(* CoDeSys 2.3.9.62 project: DrehtellerATN.pro *)
(* Libraries: Standard.lib, IecSfc.lib 2.6.14 10:37:46, SYSLIBCALLBACK.LIB *)

(* Global variable list: Global_Variables *)
VAR_GLOBAL
	Global_START: BOOL;
	K1: BOOL;
	K2: BOOL;
	Rechts: BOOL;
	Links: BOOL;
	Not_Aus: BOOL;
END_VAR

(* POU PLC_PRG, FBD *)
PROGRAM PLC_PRG
VAR
	Zweihand_Timer: TON;

END_VAR
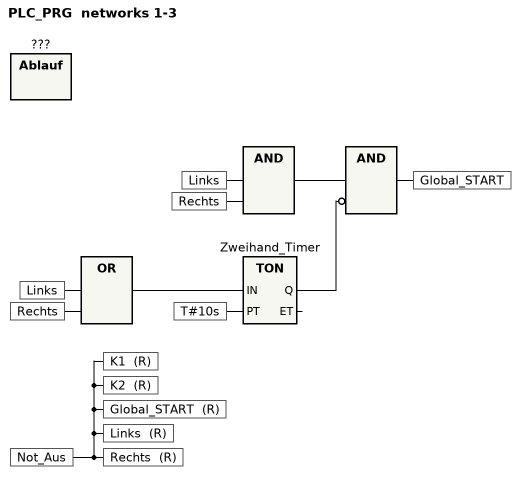
_FBD_ (* Function Block Diagram *)
NETWORK 1
	???:Ablauf()
NETWORK 2
	AND(AND(Links, Rechts), NOT Zweihand_Timer:TON(IN: OR(Links, Rechts), PT: T#10s)) => Global_START
NETWORK 3
	<<<<Not_Aus => R K1> => R K2> => R Global_START> => R Links> => R Rechts
_END_FBD_
(* the same logic as Structured Text *)
(* Network 1: see the listing above *)
(* Network 2 *)
Zweihand_Timer(IN := Links OR Rechts, PT := T#10s);
Global_START := (Links AND Rechts) AND NOT Zweihand_Timer.Q;
(* Network 3 *)
IF Not_Aus THEN K1 := FALSE; END_IF;
IF Not_Aus THEN K2 := FALSE; END_IF;
IF Not_Aus THEN Global_START := FALSE; END_IF;
IF Not_Aus THEN Links := FALSE; END_IF;
IF Not_Aus THEN Rechts := FALSE; END_IF;
END_PROGRAM

(* POU Ablauf, SFC *)
PROGRAM Ablauf
VAR
	angle:INT:=0;
	oben: BOOL:=TRUE;
	unten: BOOL;
	S1: BOOL:=TRUE;
	T1: BOOL;
	Timer1: TON;
	tor: INT;
	Rotate: BOOL:=FALSE;
END_VAR
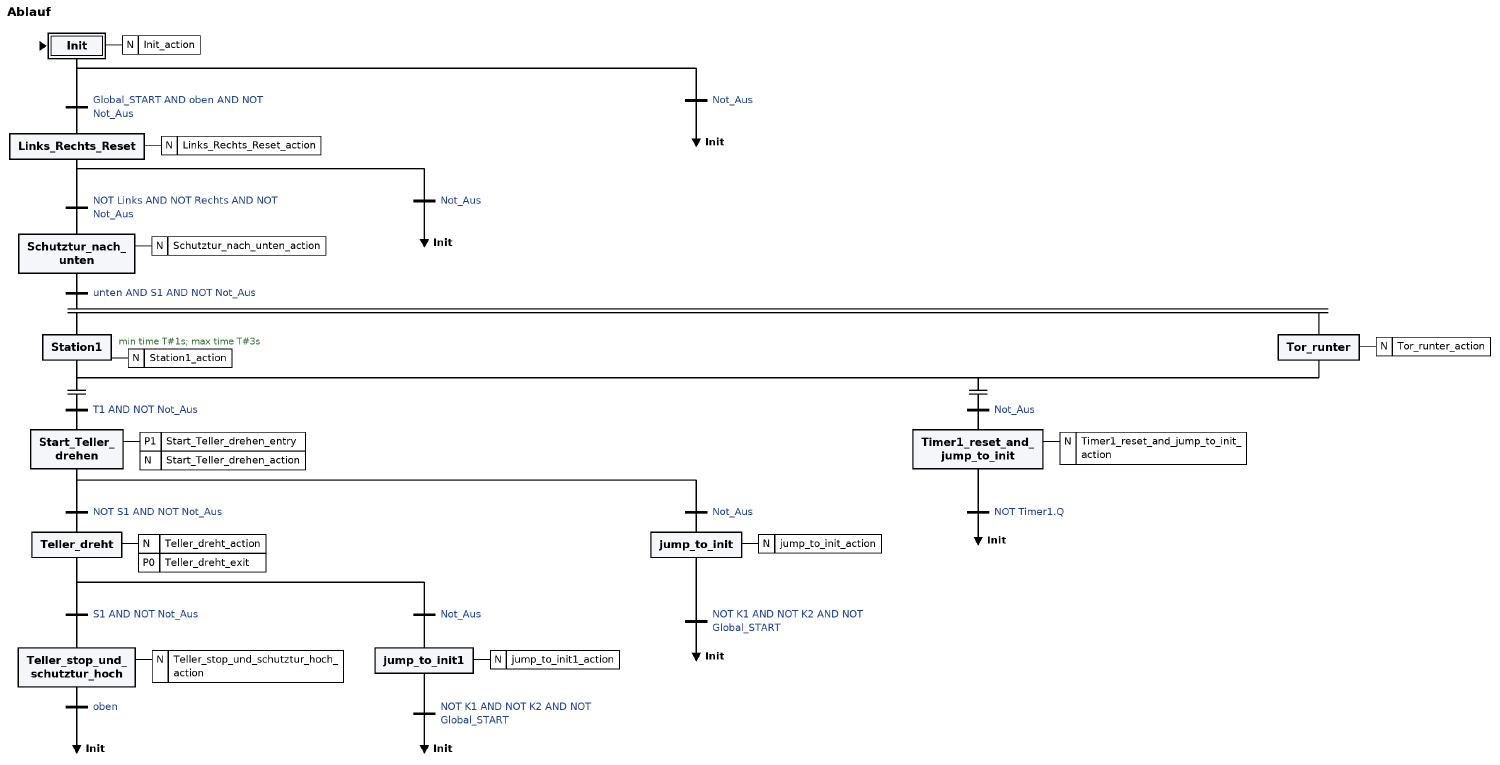
INITIAL_STEP Init:
	Init_action(N);
END_STEP
TRANSITION FROM Init TO Links_Rechts_Reset := Global_START AND oben AND NOT Not_Aus;
END_TRANSITION
TRANSITION FROM Init TO Init := Not_Aus;
END_TRANSITION
STEP Links_Rechts_Reset:
	Links_Rechts_Reset_action(N);
END_STEP
TRANSITION FROM Links_Rechts_Reset TO Schutztur_nach_unten := NOT Links AND NOT Rechts AND NOT Not_Aus;
END_TRANSITION
TRANSITION FROM Links_Rechts_Reset TO Init := Not_Aus;
END_TRANSITION
STEP Schutztur_nach_unten:
	Schutztur_nach_unten_action(N);
END_STEP
TRANSITION FROM Schutztur_nach_unten TO (Station1, Tor_runter) := unten AND S1 AND NOT Not_Aus;
END_TRANSITION
STEP Station1: (* min time T#1s; max time T#3s *)
	Station1_action(N);
END_STEP
STEP Tor_runter:
	Tor_runter_action(N);
END_STEP
TRANSITION FROM (Station1, Tor_runter) TO Start_Teller_drehen := T1 AND NOT Not_Aus;
END_TRANSITION
TRANSITION FROM (Station1, Tor_runter) TO Timer1_reset_and_jump_to_init := Not_Aus;
END_TRANSITION
STEP Timer1_reset_and_jump_to_init:
	Timer1_reset_and_jump_to_init_action(N);
END_STEP
TRANSITION FROM Timer1_reset_and_jump_to_init TO Init := NOT Timer1.Q;
END_TRANSITION
STEP Start_Teller_drehen:
	Start_Teller_drehen_entry(P1);
	Start_Teller_drehen_action(N);
END_STEP
TRANSITION FROM Start_Teller_drehen TO Teller_dreht := NOT S1 AND NOT Not_Aus;
END_TRANSITION
TRANSITION FROM Start_Teller_drehen TO jump_to_init := Not_Aus;
END_TRANSITION
STEP jump_to_init:
	jump_to_init_action(N);
END_STEP
TRANSITION FROM jump_to_init TO Init := NOT K1 AND NOT K2 AND NOT Global_START;
END_TRANSITION
STEP Teller_dreht:
	Teller_dreht_action(N);
	Teller_dreht_exit(P0);
END_STEP
TRANSITION FROM Teller_dreht TO Teller_stop_und_schutztur_hoch := S1 AND NOT Not_Aus;
END_TRANSITION
TRANSITION FROM Teller_dreht TO jump_to_init1 := Not_Aus;
END_TRANSITION
STEP jump_to_init1:
	jump_to_init1_action(N);
END_STEP
TRANSITION FROM jump_to_init1 TO Init := NOT K1 AND NOT K2 AND NOT Global_START;
END_TRANSITION
STEP Teller_stop_und_schutztur_hoch:
	Teller_stop_und_schutztur_hoch_action(N);
END_STEP
TRANSITION FROM Teller_stop_und_schutztur_hoch TO Init := oben;
END_TRANSITION

ACTION Init_action:
IF tor>0 THEN
tor:=tor-60;
S1:=TRUE;
END_IF
END_ACTION

ACTION Links_Rechts_Reset_action:
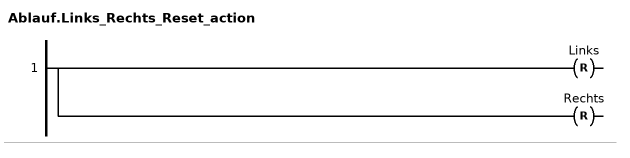
_LD_ (* Ladder Diagram *)
NETWORK 1
	* --- (R Links) (R Rechts)
_END_LD_
(* the same logic as Structured Text *)
(* Network 1 *)
Links := FALSE;
Rechts := FALSE;
END_ACTION

ACTION Schutztur_nach_unten_action:
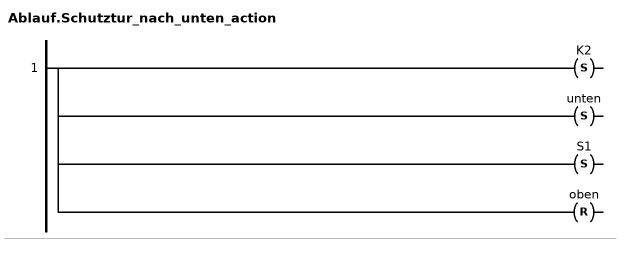
_LD_ (* Ladder Diagram *)
NETWORK 1
	* --- (S K2) (S unten) (S S1) (R oben)
_END_LD_
(* the same logic as Structured Text *)
(* Network 1 *)
K2 := TRUE;
unten := TRUE;
S1 := TRUE;
oben := FALSE;
END_ACTION

ACTION Station1_action:
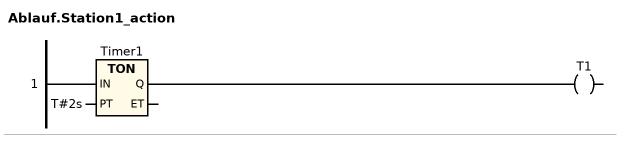
_LD_ (* Ladder Diagram *)
NETWORK 1
	Timer1:TON(IN: *, PT: T#2s) --- (T1)
_END_LD_
(* the same logic as Structured Text *)
(* Network 1 *)
Timer1(IN := TRUE, PT := T#2s);
T1 := Timer1.Q;
END_ACTION

ACTION Tor_runter_action:
IF tor=0 THEN
tor:=tor+60;
END_IF
END_ACTION

ACTION Timer1_reset_and_jump_to_init_action:
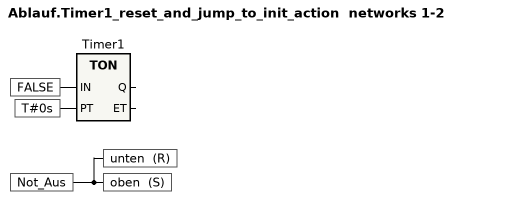
_FBD_ (* Function Block Diagram *)
NETWORK 1
	Timer1:TON(IN: FALSE, PT: T#0s)
NETWORK 2
	<Not_Aus => R unten> => S oben
_END_FBD_
(* the same logic as Structured Text *)
(* Network 1 *)
Timer1(IN := FALSE, PT := T#0s);
(* Network 2 *)
IF Not_Aus THEN unten := FALSE; END_IF;
IF Not_Aus THEN oben := TRUE; END_IF;
END_ACTION

ACTION Start_Teller_drehen_entry:
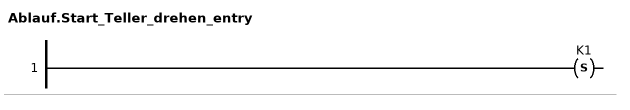
_LD_ (* Ladder Diagram *)
NETWORK 1
	* --- (S K1)
_END_LD_
(* the same logic as Structured Text *)
(* Network 1 *)
K1 := TRUE;
END_ACTION

ACTION Start_Teller_drehen_action:
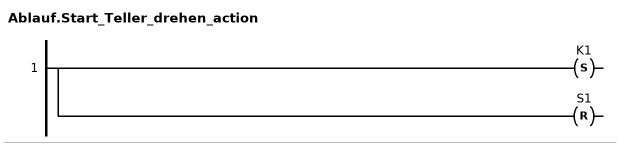
_LD_ (* Ladder Diagram *)
NETWORK 1
	* --- (S K1) (R S1)
_END_LD_
(* the same logic as Structured Text *)
(* Network 1 *)
K1 := TRUE;
S1 := FALSE;
END_ACTION

ACTION jump_to_init_action:
IF tor>0 THEN
tor:=tor-60;
S1:=TRUE;
unten:=FALSE;
oben:=TRUE;
END_IF
END_ACTION

ACTION Teller_dreht_action:
IF K1 AND NOT Rotate THEN
angle:= angle+1;
angle:= angle MOD 360;
	IF (angle MOD 90)=0 THEN
	Rotate:=TRUE;
	S1:= TRUE;
	END_IF
END_IF
END_ACTION

ACTION Teller_dreht_exit:
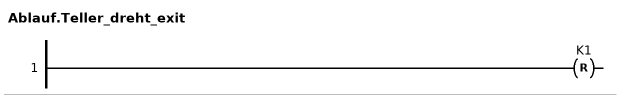
_LD_ (* Ladder Diagram *)
NETWORK 1
	* --- (R K1)
_END_LD_
(* the same logic as Structured Text *)
(* Network 1 *)
K1 := FALSE;
END_ACTION

ACTION jump_to_init1_action:
IF tor>0 THEN
tor:=tor-60;
S1:=TRUE;
unten:=FALSE;
oben:=TRUE;
END_IF
END_ACTION

ACTION Teller_stop_und_schutztur_hoch_action:
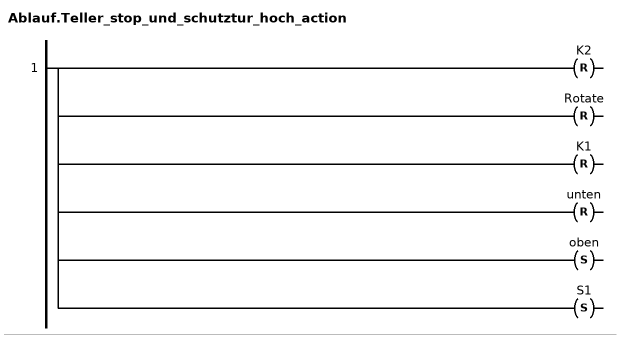
_LD_ (* Ladder Diagram *)
NETWORK 1
	* --- (R K2) (R Rotate) (R K1) (R unten) (S oben) (S S1)
_END_LD_
(* the same logic as Structured Text *)
(* Network 1 *)
K2 := FALSE;
Rotate := FALSE;
K1 := FALSE;
unten := FALSE;
oben := TRUE;
S1 := TRUE;
END_ACTION
END_PROGRAM

(* Visualisation Visalisierung
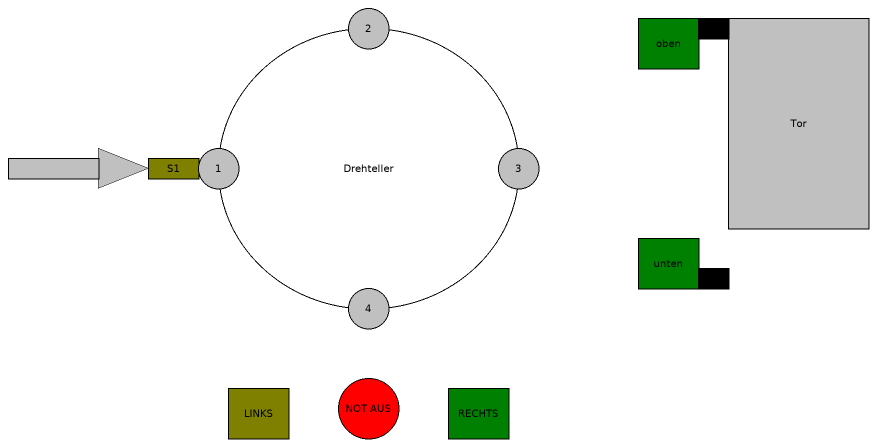
rectangle at (630,80)-(691,131): text "oben"; alarm colour if Ablauf.oben; toggles Ablauf.oben
rectangle at (140,220)-(191,241): text "S1"; alarm colour if Ablauf.S1; toggles Ablauf.S1
rectangle at (630,300)-(691,351): text "unten"; alarm colour if Ablauf.unten; toggles Ablauf.unten
ellipse at (330,440)-(391,501): text "NOT AUS"; alarm colour if .Not_Aus; toggles .Not_Aus
rectangle at (220,450)-(281,501): text "LINKS"; alarm colour if .Links; toggles .Links
rectangle at (440,450)-(501,501): text "RECHTS"; alarm colour if .Rechts; toggles .Rechts
ellipse at (210,90)-(511,371): text "Drehteller"
ellipse at (190,210)-(231,251): text "1"; angle Ablauf.angle
ellipse at (340,70)-(381,111): text "2"; angle Ablauf.angle
ellipse at (490,210)-(531,251): text "3"; angle Ablauf.angle
ellipse at (340,350)-(381,391): text "4"; angle Ablauf.angle
rectangle at (720,80)-(861,291): text "Tor"; y offset Ablauf.tor
4 more shapes without text or variables
*)
